# EPICS autosave request: iocBoot/ioc13Raman2/auto_settings.req
file "userArrayCalcs10_settings.req",   P=$(P)
file "userCalcOuts10_settings.req",     P=$(P)
file "userStringCalcs10_settings.req",  P=$(P)
file "userStringSeqs10_settings.req",   P=$(P)
file "userTransforms10_settings.req",   P=$(P)
file "scan_settings.req",               P=$(P), S=scan1
file "scan_settings.req",               P=$(P), S=scan2
file "scan_settings.req",               P=$(P), S=scan3
file "scan_settings.req",               P=$(P), S=scan4
file "CARS_motor_settings.req",         P=$(P), M=m1
file "CARS_motor_settings.req",         P=$(P), M=m2
file "CARS_motor_settings.req",         P=$(P), M=m3
file "CARS_motor_settings.req",         P=$(P), M=m4
file "CARS_motor_settings.req",         P=$(P), M=m5
file "CARS_motor_settings.req",         P=$(P), M=m6
file "CARS_motor_settings.req",         P=$(P), M=m7
#file "CARS_motor_settings.req",         P=$(P), M=m9
#file "CARS_motor_settings.req",         P=$(P), M=m10
#file "CARS_motor_settings.req",         P=$(P), M=m11
#file "CARS_motor_settings.req",         P=$(P), M=m12
#file "CARS_motor_settings.req",         P=$(P), M=m13
#file "CARS_motor_settings.req",         P=$(P), M=m14
#file "CARS_motor_settings.req",         P=$(P), M=m15
file "saveData_settings.req"            P=$(P)
